Universal Robots PolyScope program: clawMarchine.urp

Program clawMarchine (installation=default directory=/programs/usbdisk/2023 createdIn=5.11.10.1010502 lastSavedIn=5.11.10.1010502 robotSerialNumber=20205300125)
Calibrated DH parameters: a=[-0.000042, -0.183432, -0.213066, 0.000185, -0.000084, 0]; d=[0.152126, -129.800832, 134.536465, -4.604531, 0.085429, 0.092211]; alpha=[1.571458, -0.001234, 0.002522, 1.571667, -1.572664, 0]; deltaTheta=[0, 0.717739, -0.661739, -0.056003, -0.000002, 0]
BeforeStart
  var_p := p_start
  MoveJ speed 60 deg/s, acceleration 80 deg/s^2 (useActiveTCP=true) feature=Base
    Waypoint p_start: TCP in base x=0.011 y=-300.005 z=200.01 mm, rx=0.1509 ry=3.1379 rz=0 rad; joints [-64.138, -89.857, -60.376, -119.659, 90.134, 31.394] deg
    URCap RG 그립 (OnRobot, OnRobot A/S) dataModel(rg-target-force=40.0, rg-target-width=0.005)
Robot Program (runOnlyOnce=false)
  Switch expression=read_port_register(130)
    Case (caseValue=1)
      Script: var_p=pose_add(get_actual_tcp_pose(), p[0,0.3,0,0,0,0])
      MoveL speed 100 mm/s, acceleration 600 mm/s^2 (useActiveTCP=true) feature=Base
        Waypoint 웨이포인트 (Variable): variable=var_p
          Until EXPRESSION (allowActions=false) ExpressionBranch=read_port_register(130)≟0
    Case (caseValue=2)
      Script: var_p=pose_add(get_actual_tcp_pose(), p[-0.3,0,0,0,0,0])
      MoveL speed 100 mm/s, acceleration 600 mm/s^2 (useActiveTCP=true) feature=Base
        Waypoint 웨이포인트 (Variable): variable=var_p
          Until EXPRESSION (allowActions=false) ExpressionBranch=read_port_register(130)≟0
    Case (caseValue=3)
      Script: var_p=pose_add(get_actual_tcp_pose(), p[0,-0.3,0,0,0,0])
      MoveL speed 100 mm/s, acceleration 600 mm/s^2 (useActiveTCP=true) feature=Base
        Waypoint 웨이포인트 (Variable): variable=var_p
          Until EXPRESSION (allowActions=false) ExpressionBranch=read_port_register(130)≟0
    Case (caseValue=4)
      Script: var_p=pose_add(get_actual_tcp_pose(), p[0.3,0,0,0,0,0])
      MoveL speed 100 mm/s, acceleration 600 mm/s^2 (useActiveTCP=true) feature=Base
        Waypoint 웨이포인트 (Variable): variable=var_p
          Until EXPRESSION (allowActions=false) ExpressionBranch=read_port_register(130)≟0
    Case (caseValue=5)
      var_p := get_actual_tcp_pose()
      URCap RG 그립 (OnRobot, OnRobot A/S) dataModel(rg-target-force=40.0, rg-target-width=0.07)
      Script: zero_ftsensor()
      Force Simple feature=Base; selection=[0, 0, 1, 0, 0, 0]; wrench=[0, 0, -3, 0, 0, 0]; limitsForce=[0.15, 0.15, 0.15, 1.047198, 1.047198, 1.047198]; limitsMotion=[0.1, 0.1, 0.1, 0.349066, 0.349066, 0.349066]
        Wait Condition expression=force()≥10
        URCap RG 그립 (OnRobot, OnRobot A/S) dataModel(rg-target-force=40.0, rg-target-width=0.005, Variable(key=on_return, variable(name=on_return)))
      MoveL speed 250 mm/s, acceleration 1200 mm/s^2 (useActiveTCP=true) feature=Base
        Waypoint 웨이포인트 (Variable): variable=var_p
        Script: write_port_register(130,0)
      MoveJ speed 60 deg/s, acceleration 80 deg/s^2 (useActiveTCP=true) feature=Base
        Waypoint p_dropUp: TCP in base x=0.005 y=-390.347 z=199.992 mm, rx=0.151 ry=3.1379 rz=0.0001 rad; joints [-70.408, -119.212, -20.844, -129.84, 90.085, 25.121] deg
      MoveL speed 250 mm/s, acceleration 1200 mm/s^2 (useActiveTCP=true) feature=Base
        Script: zero_ftsensor()
        Force Simple feature=Base; selection=[0, 0, 1, 0, 0, 0]; wrench=[0, 0, -3, 0, 0, 0]; limitsForce=[0.15, 0.15, 0.15, 1.047198, 1.047198, 1.047198]; limitsMotion=[0.1, 0.1, 0.1, 0.349066, 0.349066, 0.349066]
          Wait Condition expression=force()≥10
          URCap RG 그립 (OnRobot, OnRobot A/S) dataModel(rg-target-force=40.0, rg-target-width=0.07, Variable(key=on_return, variable=on_return))
        Waypoint p_dropUp: TCP in base x=0.005 y=-390.347 z=199.992 mm, rx=0.151 ry=3.1379 rz=0.0001 rad; joints [-70.408, -119.212, -20.844, -129.84, 90.085, 25.121] deg
      MoveJ speed 60 deg/s, acceleration 80 deg/s^2 (useActiveTCP=true) feature=Base
        Waypoint p_start referenceName=p_start: TCP in base x=0.011 y=-300.005 z=200.01 mm, rx=0.1509 ry=3.1379 rz=0 rad; joints [-64.138, -89.857, -60.376, -119.659, 90.134, 31.394] deg
    Case (caseValue=6)
      var_p := pose_trans(get_actual_tcp_pose(),p[0,0,0,0,0,-3.14] )
      MoveL speed 250 mm/s, acceleration 1200 mm/s^2 (useActiveTCP=true) feature=Base
        Waypoint 웨이포인트 (Variable): variable=var_p
          Until EXPRESSION (allowActions=false) ExpressionBranch=read_port_register(130)≟0
    Case (caseValue=7)
      var_p := pose_trans(get_actual_tcp_pose(),p[0,0,0,0,0,3.14] )
      MoveL speed 250 mm/s, acceleration 1200 mm/s^2 (useActiveTCP=true) feature=Base
        Waypoint 웨이포인트 (Variable): variable=var_p
          Until EXPRESSION (allowActions=false) ExpressionBranch=read_port_register(130)≟0
